FUNCTION F_GetDistToPosModulo : LREAL //This is only working in Positiv Direktion
VAR_INPUT
	fTargetPosition : LREAL;
	fActualPosition : LREAL;
	fModulo 		: LREAL;
END_VAR

VAR

END_VAR

IF fTargetPosition < fActualPosition THEN
	fTargetPosition := fTargetPosition + fModulo;
END_IF

F_GetDistToPosModulo := fTargetPosition - fActualPosition;

END_FUNCTION

(* stored: Version 1.1.0.1, ProductVersion 3.1.4024.15
   POU F_GetDistToPosModulo: Id {9aca93c6-8bd8-4f96-89e8-11b79549961d}, SpecialFunc None *)
